//The Timing Analysis 1Ch measures time difference between on- and off-periods and counts the amount of on-periods. The on-period starts when the condition of operator and threshold is met. Optional a boolean signal for Enable Execution can be selected, so that the algorithm is just active if the value of the selected signal is TRUE.
FUNCTION_BLOCK FB_N1_M3_State_Aborted
VAR_INPUT
	nDataIn: UINT; 
	tTimestamp: ULINT; 
	bEnableExecution: BOOL := TRUE; 
	bReset: BOOL; 
	bReconfigure: BOOL := TRUE;
END_VAR
VAR_INPUT PERSISTENT
	stThresholdLevelOn: ST_ALY_Threshold; 
	fTolerance: LREAL; 
END_VAR
VAR_OUTPUT
	bError: BOOL;
	ipTcResult: I_TcMessage;
	bNewResult: BOOL;
	bIsOn: BOOL;
	nCountOn: ULINT;
	fbTimeCurrentInterval: FB_ALY_TimeSpan;
	fbTimeOnTotal: FB_ALY_TimeSpan;
	fbTimeOffTotal: FB_ALY_TimeSpan;
END_VAR
VAR
	
	R_TRIG_Reconfigure: R_TRIG;
	
	fbALY_TimingAnalysis_1Ch: FB_ALY_TimingAnalysis_1Ch := ( bPersistent:= TRUE );
END_VAR
VAR PERSISTENT
	bConfigured: BOOL;
END_VAR

METHOD Call : BOOL
VAR_INPUT
	nCurrentContext: DWORD;
END_VAR
VAR
END_VAR
IF NOT bConfigured THEN
	bConfigured:= TRUE;

	fTolerance:= 0;

	stThresholdLevelOn.eComparisonOperator:= E_ALY_ComparisonOperator.Equals;
	stThresholdLevelOn.fThreshold:= 9;

	fbALY_TimingAnalysis_1Ch.fTolerance:= fTolerance;
END_IF

R_TRIG_Reconfigure(CLK:= bReconfigure);
IF R_TRIG_Reconfigure.Q THEN
	fbALY_TimingAnalysis_1Ch.ConfigureChannel(stThresholdLevel:= stThresholdLevelOn);

	fbALY_TimingAnalysis_1Ch.Configure();

	bReconfigure:= FALSE;
END_IF

IF bReset THEN
	Reset();
END_IF

IF bEnableExecution THEN
	IF F_HasContext(nCurrentContext, nContext) THEN
		fbALY_TimingAnalysis_1Ch.SetChannelValue(Input:= nDataIn);

		fbALY_TimingAnalysis_1Ch.Call(tTimestamp:= tTimestamp);

		bNewResult:= fbALY_TimingAnalysis_1Ch.bNewResult;
		bIsOn:= fbALY_TimingAnalysis_1Ch.bIsOn;
		nCountOn:= fbALY_TimingAnalysis_1Ch.nCountOn;
		fbTimeCurrentInterval:= fbALY_TimingAnalysis_1Ch.fbTimeCurrentInterval;
		fbTimeOnTotal:= fbALY_TimingAnalysis_1Ch.fbTimeOnTotal;
		fbTimeOffTotal:= fbALY_TimingAnalysis_1Ch.fbTimeOffTotal;

		bError:= fbALY_TimingAnalysis_1Ch.bError;
		ipTcResult:= fbALY_TimingAnalysis_1Ch.ipResultMessage;
	END_IF
ELSE
	bNewResult:= FALSE;
END_IF
END_METHOD

METHOD Reset : BOOL
VAR
END_VAR
Reset:= fbALY_TimingAnalysis_1Ch.Reset();

bNewResult:= fbALY_TimingAnalysis_1Ch.bNewResult;
bIsOn:= fbALY_TimingAnalysis_1Ch.bIsOn;
nCountOn:= fbALY_TimingAnalysis_1Ch.nCountOn;
fbTimeCurrentInterval:= fbALY_TimingAnalysis_1Ch.fbTimeCurrentInterval;
fbTimeOnTotal:= fbALY_TimingAnalysis_1Ch.fbTimeOnTotal;
fbTimeOffTotal:= fbALY_TimingAnalysis_1Ch.fbTimeOffTotal;

bError:= NOT Reset;
ipTcResult:= fbALY_TimingAnalysis_1Ch.ipResultMessage;
END_METHOD

PROPERTY nContext : DWORD
GET
nContext:= E_VirtualInput.eContext_V1_Virtual_Input_Source;
END_GET
END_PROPERTY

END_FUNCTION_BLOCK

(* stored: POU FB_N1_M3_State_Aborted: Id 0330c632-6883-4287-8677-d13016a5520c, SpecialFunc None
   Method Call: Id bfe09ca3-1bd5-44b5-abf1-0a1f5aa22d6c
   Method Reset: Id 6dcae22d-7df6-4288-a09b-62afabd61420
   Property nContext: Id 561a350a-99e8-4b58-ab86-7e96a0242db5
   Get Get: Id 7bce6e94-d962-487a-86a3-27abec792589 *)
